// TIA Portal V16 export
// export: Created 2021-09-08T12:46:11.9565367Z, ExportSetting WithDefaults, DisplayName Totally Integrated Automation Portal, DisplayVersion V16 Update 3, DisplayName TIA Portal Version Control Interface, DisplayVersion V16 Update 2, DisplayName TIA Portal Openness, DisplayVersion V16 Update 3, DisplayName TIA Portal Teamcenter Gateway, DisplayVersion V16, DisplayName STEP 7 Professional, DisplayVersion V16 Update 3, DisplayName STEP 7 Safety, DisplayVersion V16, DisplayName WinCC Advanced, DisplayVersion V16 Update 3
DATA_BLOCK "dtPumpSetup"   // DB5
{ S7_Optimized_Access := 'FALSE' }
VERSION : 0.1
// stored: AutoNumber true, DBAccessibleFromOPCUA true, IsOnlyStoredInLoadMemory false, IsWriteProtectedInAS false
   VAR RETAIN
      modeP30x : Bool;
      cmStartP30x : Bool;
      selectP30x { S7_SetPoint := 'True'} : Bool;
      freqStopP30x { S7_SetPoint := 'True'} : Real := 31.0;
      delayStopP30x { S7_SetPoint := 'True'} : Real := 5.0;
      presStartP30x { S7_SetPoint := 'True'} : Real := 2.0;
      delayStartP30x { S7_SetPoint := 'True'} : Real := 1.0;
      levTW20xStartP30x { S7_SetPoint := 'True'} : Real := 30.0;
      levTW20xStopP30x { S7_SetPoint := 'True'} : Real := 10.0;
      modeP120x : Bool;
      cmStartP120x : Bool;
      selectP120x { S7_SetPoint := 'True'} : Bool;
      timeNoPulseP120x { S7_SetPoint := 'True'} : Real := 31.0;
      presStartP120x { S7_SetPoint := 'True'} : Real := 2.0;
      delayStartP120x { S7_SetPoint := 'True'} : Real := 1.0;
      levTW11xStartP120x { S7_SetPoint := 'True'} : Real := 30.0;
      levTW11xStopP120x { S7_SetPoint := 'True'} : Real := 10.0;
      modeP150x : Bool;
      cmStartP150x : Bool;
      selectP150x { S7_SetPoint := 'True'} : Bool;
      timeNoPulseP150x { S7_SetPoint := 'True'} : Real := 31.0;
      presStartP150x { S7_SetPoint := 'True'} : Real := 2.0;
      delayStartP150x { S7_SetPoint := 'True'} : Real := 1.0;
      levTW14xStartP150x { S7_SetPoint := 'True'} : Real := 30.0;
      levTW14xStopP150x { S7_SetPoint := 'True'} : Real := 10.0;
      tChangeP30x { S7_SetPoint := 'True'} : Real := 12.0;
      tChangeP120x { S7_SetPoint := 'True'} : Real := 12.0;
      tChangeP150x { S7_SetPoint := 'True'} : Real := 12.0;
      tToChangeP30x : Real;
      tToChangeP120x : Real;
      tToChangeP150x : Real;
      modeP70x : Bool;
      cmP70x : Bool;
      selectP70x : Bool;
      tChangeP70x { S7_SetPoint := 'True'} : Real := 24.0;
      tToChangeP70x : Real;
   END_VAR
BEGIN
END_DATA_BLOCK
